{attribute addProperty BoxType "EJ1914-0000-0017"}
{attribute addProperty Id "Fieldvoltage_UnderrangeAT %I*BOOL811Fieldvoltage_OverrangeAT %I*BOOL812"}
{attribute addProperty CRC "3401588706"}
{attribute addProperty SizeInBites "16"}
{attribute addProperty SizeInBytes "2"}
TYPE FIELDVOLTAGE_Field_Voltage_Status_CAC01FE2 :
STRUCT
	{attribute addProperty Name "Fieldvoltage_Underrange"}
	Fieldvoltage_Underrange AT %I* : BOOL;
	{attribute addProperty Name "Fieldvoltage_Overrange"}
	Fieldvoltage_Overrange AT %I* : BOOL;
END_STRUCT
END_TYPE

(* stored: Version 1.2.0.0, ProductVersion 3.1.4024.9
   DUT FIELDVOLTAGE_Field_Voltage_Status_CAC01FE2: Id {20cc00a6-4957-425e-9789-39b1d37c3752} *)
